PROGRAM MAIN
VAR
	Waarde: BYTE;
	potentiometer: INT;
END_VAR

(*
Potentiometer inlezen (maximaal 1 regels)

Lees de potentiometer in en verschaal deze waarden naar een getal tussen 0 en 100.
*)
Waarde:=LREAL_TO_BYTE(100*(potentiometer/32767.0));

END_PROGRAM

(* stored: Version 1.1.0.1, ProductVersion 3.1.4024.12
   POU MAIN: Id {dbd9d2a5-fc61-49b0-b1c6-67cdcddd58c8}, SpecialFunc None *)
